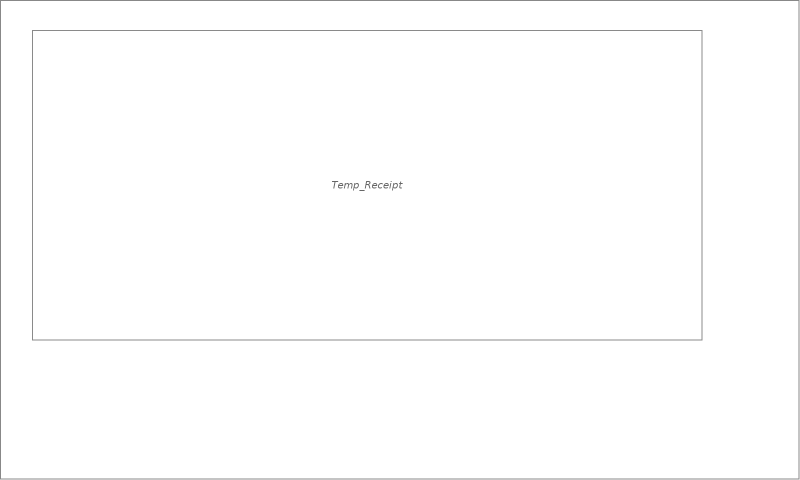
VISUALIZATION Visu_ReceiptList_01  // 800x480
    Frame (32,30 670x310)
        shows Temp_Receipt(stHmiRData := stRData[1])
END_VISUALIZATION

(* stored: Version 1.1.0.1, ProductVersion 3.1.4024.6
   Visu Visu_ReceiptList_01: Id {0797afca-8c78-48af-a7e5-d9762e946906} *)
